Yaskawa INFORM job: POUNCE.JBI

/JOB
//NAME POUNCE
///FOLDERNAME SPEEDBOT
//POS
///NPOS 1,0,0,0,0,0
///TOOL 0
///POSTYPE PULSE
///PULSE
C00000=21627,0,0,0,0,0
//INST
///DATE 2024/08/21 10:14
///COMM V0.1
///ATTR SC,RW
///GROUP1 RB1
NOP
'*********************
'POUNCE
'*********************
'发送路径号 1
MACRO1 MJ#(1) ARGF1
'示教 POUNCE 位置
MOVJ C00000 VJ=80.00
MACRO1 MJ#(0)
SET B001 B000
'当路径号为 255 时返回原点
IFTHENEXP B000=255
MACRO1 MJ#(1) ARGF2
CALL JOB:MOVE_TO_HOME
ABORT
ENDIF
END
